PROGRAM P_Demo_FB_DMXSetLampHours
VAR
    fbSetLampHours    : FB_DMXSetLampHours;           // 写灯泡点亮小时数
    stDmxCmdBuffer    : ST_DMXCommandBuffer;          // 与通讯 FB 共用
    wTargetManufId    : WORD := 16#4241;              // 目标灯具厂商 ID
    dwTargetDeviceId  : DWORD := 16#12131415;         // 目标灯具设备 ID
    byTargetPort      : BYTE := 0;                    // 根设备通道 0
    udiNewHours       : UDINT := 0;                   // 换灯后清零
    bDoSet            : BOOL := FALSE;                // 在线给一次上升沿触发
    bBusy             : BOOL;
    bError            : BOOL;
    udiErrId          : UDINT;
END_VAR

// ============================================================
// Tc2_DMX.FB_DMXSetLampHours 演示程序
// ============================================================
// 场景：灯泡更换作业：换新灯后把该灯具点亮小时计数器清零，寿命统计从 0 重新开始。
// 价值：把换灯后的计数器复位做成一次 PLC 调用，保证寿命管理数据与实际灯泡同步。
// 验证：设 udiNewHours:=0，给 bDoSet 一次上升沿 -> bBusy 短暂 TRUE -> 回 FALSE 后用 FB_DMXGetLampHours 回读应为 0。
// 验证步骤：
//   1. 右键 PLC 项目下 POUs 文件夹 → Add → Existing Item → 选本 .TcPOU 文件
//   2. 引用 Tc2_DMX；同项目里放一个 FB_EL6851CommunicationEx 实例并共用 stDmxCmdBuffer（非 CycleMode）
//   3. 编译 → 登录 → 运行；按上方『验证』行在线给上升沿观察
// ============================================================

fbSetLampHours(
    bStart                     := bDoSet,
    wDestinationManufacturerId := wTargetManufId,
    dwDestinationDeviceId      := dwTargetDeviceId,
    byPortId                   := byTargetPort,
    udiLampHours               := udiNewHours,
    dwOptions                  := 0,
    stCommandBuffer            := stDmxCmdBuffer,
    bBusy                      => bBusy,
    bError                     => bError,
    udiErrorId                 => udiErrId
);

END_PROGRAM

(* stored: Version 1.1.0.1, ProductVersion 3.1.4024.5
   POU P_Demo_FB_DMXSetLampHours: Id {5cab4a5a-f7fa-513c-88ad-7823b262ffa3}, SpecialFunc None *)
